Staubli VAL3: Bewegungsattribute.dtx

frame StaubliTX240Base = {x=0.000, y=0.000, z=0.000, rx=-0.000, ry=0.000, rz=-0.000, fatherId=world[0]}
tool tCurrentTool = {x=0.000, y=0.000, z=0.000, rx=-0.000, ry=0.000, rz=-0.000, fatherId=flange[0]}
mdesc mCurrentSpeed
pointRx pPointRx1 = {}
pointRx pPointRx2 = {}
